TYPE DUT_ChangeBatchPositionInProductionQueue:
STRUCT  
	return_value		: DINT;
	BatchId				: STRING(50);
	DestinationPosition : DINT;
END_STRUCT
END_TYPE

(* stored: Version 1.1.0.1, ProductVersion 3.1.4024.15
   DUT DUT_ChangeBatchPositionInProductionQueue: Id {cf8583ed-3a60-43eb-ade5-3e80ef6c71eb} *)
